TYPE (* IEC61131-3, Table 14#5 *)
  (* Standard: 1131-3 *)
  (* Version 0.0, 1/8/2024, Cheyan, Schneider Electric, Template *)
  PACKAGE Main;
  {SET_ATTRIBUTE(nxtDataType, p1MX6tImGfRGisjIz/Bb0Mcm6lYG2l98Aoeyk/36Lw1UnDbkGzeKcJs8tmta5EK7GSMGtmwYiPA=)}
  source : (
    process,
    substituted,
    process
  );
END_TYPE
